{attribute 'Tc2GvlVarNames'}
{attribute 'strict'}
//Tipologia di "Pallet/Cassa/Cavalletto" 
TYPE e_Tipo_Pallet :
(
	NOT_DEFINED			:= 0,
	PALLET_STANDARD 	:= 1, (* Indica la tipologia di Pallet standard *)
	CASSA_STANDARD		:= 2,(* Indica la tipologia di cassa in legno standard *)
	CAVALLETTO			:= 3,(* Indica la tipologia cavalletto GENERICA *)
	PALLET_ACCOPPIATI 	:= 4, (* Indica la tipologia di Pallet standard ACCOPPIATI A 2 *)
	BUNDLE				:= 5,  (* Indica la tipologia di Cavallina ad un solo lato *)
	PIANALE_GENERICO	:= 6, (* Indica un pianale generico *)
	ELEMENTO_PIANO_GENERICO := 10, (* Indica un elemento piano generico, ovvero palleto, cassa, pianale,ecc*)
	ELEMENTO_VERT_GENERICO := 11 (* Indica un elemento verticale generico, ovvero A-Frame-Bundle *)
);
END_TYPE

(* stored: Version 1.1.0.1, ProductVersion 3.1.4024.11
   EnumerationTextList e_Tipo_Pallet: Id {99c47fc9-51a1-4b62-8af3-0306c28f18ae} *)
